FUNCTION_BLOCK EtherNetIPMaster
VAR_INPUT
END_VAR
VAR_OUTPUT
END_VAR
VAR
	DevState AT%i* : UINT;
END_VAR

END_FUNCTION_BLOCK

(* stored: Version 1.1.0.1, ProductVersion 3.1.4024.11
   POU EtherNetIPMaster: Id {23d346be-69ba-4116-9848-11de21f5338e}, SpecialFunc None *)
